// Mitsubishi GX Works2 project: n02   PLC: Q02/Q02H

PROGRAM MAIN
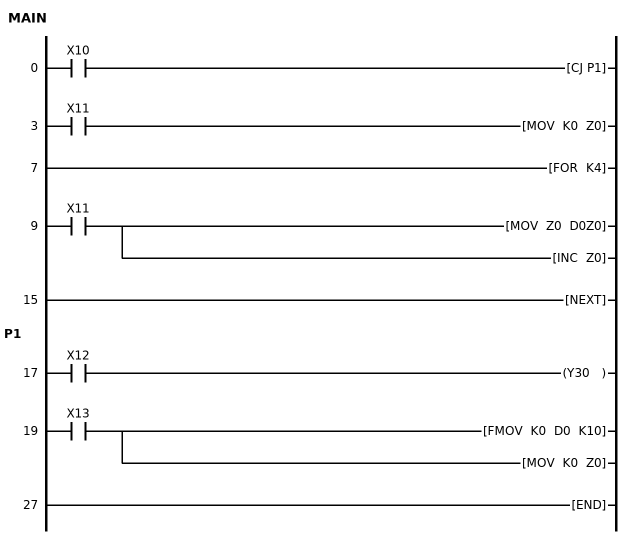
0     LD      X10
      CJ      P1
3     LD      X11
      MOV     K0 Z0
7     FOR     K4
9     LD      X11
      MOV     Z0 D0Z0
      INC     Z0
15    NEXT
      P1
17    LD      X12
      OUT     Y30
19    LD      X13
      FMOV    K0 D0 K10
      MOV     K0 Z0
27    END
END_PROGRAM
